{attribute 'linkalways'} 
{attribute 'no_explicit_call' := 'This FB is a CLASS and must be accessed using methods or properties'}
FUNCTION_BLOCK Nci EXTENDS CyclicInstance IMPLEMENTS I_Nci
VAR
	_nciPlc : NciPlc;
END_VAR

PROPERTY _InternalNciPlcRef : REFERENCE TO NciPlc
GET
_InternalNciPlcRef REF= _nciPlc;
END_GET
END_PROPERTY

METHOD AddAxisToGroup
VAR_INPUT
	axis : I_Axis;
	index : UDINT;
	timeout : TIME;
	feedback : REFERENCE TO I_CommandFeedback;
END_VAR
VAR_INST
	pCmd : POINTER TO AddAxisToGroupCommand;
END_VAR
VAR
	_axis : I_Axis;
	_index : UDINT;
	_timeout : TIME;
END_VAR
_axis := axis;
_index := index;
_timeout := timeout;

pCmd := __NEW(AddAxisToGroupCommand(
	nci := THIS^,
	axis := _axis,
	index := _index,
	timeout := _timeout
));

(*
This doesn't work hence the horrible hack with intermediate values

pCmd := __NEW(AddAxisToGroupCommand(
	nci := THIS^,
	axis := axis,
	index := index,
	timeout := timeout
));
*)

pCmd^.Execute(feedback).ThenRelease();
END_METHOD

PROPERTY BlockNumber : UDINT
GET
BlockNumber := ItpGetBlockNumber(THIS^._nciPlc.nciToPlc);
END_GET
END_PROPERTY

METHOD BuildXYGroup
VAR_INPUT
	xAxis : I_Axis;
	yAxis : I_Axis;
	timeout : TIME;
	feedback : REFERENCE TO I_CommandFeedback;
END_VAR
VAR
	null : I_Axis;
END_VAR
BuildXYZGroup(xAxis, yAxis, null, timeout, feedback);
END_METHOD

METHOD BuildXYZGroup
VAR_INPUT
	xAxis : I_Axis;
	yAxis : I_Axis;
	zAxis : I_Axis;
	timeout : TIME;
	feedback : REFERENCE TO I_CommandFeedback;
END_VAR
VAR_INST
	pCmd : POINTER TO BuildXYZGroupCommand;
END_VAR
VAR
	_xAxis : I_Axis;
	_yAxis : I_Axis;
	_zAxis : I_Axis;
	_timeout : TIME;
END_VAR
_xAxis := xAxis;
_yAxis := yAxis;
_zAxis := zAxis;
_timeout := timeout;

pCmd := __NEW(BuildXYZGroupCommand(
	nci := THIS^,
	xAxis := _xAxis,
	yAxis := _yAxis,
	zAxis := _zAxis,
	timeout := _timeout
));

(*
This doesn't work hence the horrible hack with intermediate values

pCmd := __NEW(BuildXYZGroupCommand(
	nci := THIS^,
	xAxis := xAxis,
	yAxis := yAxis,
	zAxis := zAxis,
	timeout := commandTimeout
));
*)

pCmd^.Execute(feedback).ThenRelease();
END_METHOD

PROPERTY ChannelId : UINT
GET
ChannelId := ItpGetChannelId(THIS^._nciPlc.nciToPlc);
END_GET
END_PROPERTY

PROPERTY ChannelType : ChannelType
GET
VAR
	inter : INT;
	pInter : POINTER TO ChannelType;
END_VAR
// Don't know how to do the type conversion with NCIChannelType being strict
inter := ItpGetChannelType(THIS^._nciPlc.nciToPlc);
pInter := ADR(inter);
ChannelType := pInter^;
END_GET
END_PROPERTY

METHOD  CyclicCall
END_METHOD

PROPERTY ErrorId : UDINT
GET
ErrorId := ItpGetError(THIS^._nciPlc.nciToPlc);
END_GET
END_PROPERTY

METHOD GetGroupAxisIds : DWORD
VAR_IN_OUT
	axisIds : ARRAY[1..8] OF DWORD;
END_VAR
GetGroupAxisIds := ItpGetGroupAxisIds(axisIds, THIS^._nciPlc.nciToPlc);
END_METHOD

METHOD GetOverride : LREAL
GetOverride := ItpGetOverridePercent(THIS^._nciPlc.plcToNci);
END_METHOD

PROPERTY GroupId : UDINT
GET
GroupId := ItpGetGroupId(THIS^._nciPlc.nciToPlc);
END_GET
END_PROPERTY

PROPERTY HandshakeableMFunction : INT
GET
HandshakeableMFunction := ItpGetHskMFunc(THIS^._nciPlc.nciToPlc);
END_GET
END_PROPERTY

PROPERTY HasError : BOOL
GET
HasError := ItpHasError(THIS^._nciPlc.nciToPlc);
END_GET
END_PROPERTY

PROPERTY HParam : DINT
GET
HParam := ItpGetHParam(THIS^._nciPlc.nciToPlc);
END_GET
END_PROPERTY

PROPERTY InterpreterState : UDINT
GET
InterpreterState := ItpGetStateInterpreter(THIS^._nciPlc.nciToPlc);
END_GET
END_PROPERTY

PROPERTY IsEstop : BOOL
GET
IsEstop := ItpIsEStopEx(THIS^._nciPlc.nciToPlc);
END_GET
END_PROPERTY

METHOD IsFastMFunctionPresent : BOOL
VAR_INPUT
	functionNumber : INT;
END_VAR
IsFastMFunctionPresent := ItpIsFastMFunc(functionNumber, THIS^._nciPlc.nciToPlc);
END_METHOD

METHOD IsHandshakeableMFunctionPresent : BOOL
IsHandshakeableMFunctionPresent := ItpIsHskMFunc(THIS^._nciPlc.nciToPlc);
END_METHOD

METHOD ReadCyclicLRealParameter : LREAL
VAR_INPUT
	parameterNumber : UINT(1..4);
END_VAR
CASE parameterNumber OF
	1: ReadCyclicLRealParameter := ItpReadCyclicLRealParam1(THIS^._nciPlc.nciToPlc);
	2: ReadCyclicLRealParameter := ItpReadCyclicLRealParam2(THIS^._nciPlc.nciToPlc);
	3: ReadCyclicLRealParameter := ItpReadCyclicLRealParam3(THIS^._nciPlc.nciToPlc);
	4: ReadCyclicLRealParameter := ItpReadCyclicLRealParam4(THIS^._nciPlc.nciToPlc);
END_CASE
END_METHOD

METHOD ReadCyclicUdintParameter : UDINT
VAR_INPUT
	parameterNumber : UINT(1..4);
END_VAR
CASE parameterNumber OF
	1: ReadCyclicUdintParameter := ItpReadCyclicUdintParam1(THIS^._nciPlc.nciToPlc);
	2: ReadCyclicUdintParameter := ItpReadCyclicUdintParam2(THIS^._nciPlc.nciToPlc);
	3: ReadCyclicUdintParameter := ItpReadCyclicUdintParam3(THIS^._nciPlc.nciToPlc);
	4: ReadCyclicUdintParameter := ItpReadCyclicUdintParam4(THIS^._nciPlc.nciToPlc);
END_CASE
END_METHOD

METHOD ReleaseAxis
VAR_INPUT
	axis : I_Axis;
	timeout : TIME;
	feedback : REFERENCE TO I_CommandFeedback;
END_VAR
VAR_INST
	pCmd : POINTER TO ReleaseAxisCommand;
END_VAR
VAR
	_axis : I_Axis;
	_timeout : TIME;
END_VAR
_axis := axis;
_timeout := timeout;

pCmd := __NEW(ReleaseAxisCommand(
	axis := _axis,
	timeout := _timeout
));

(*
This doesn't work hence the horrible hack with intermediate values

pCmd := __NEW(ReleaseAxisCommand(
	axis := axis,
	timeout := timeout
));
*)
pCmd^.Execute(feedback).ThenRelease();
END_METHOD

METHOD ResetGroup
VAR_INPUT
	timeout : TIME;
	feedback : REFERENCE TO I_CommandFeedback;
END_VAR
VAR_INST
	pCmd : POINTER TO ResetGroupCommand;
END_VAR
VAR
	_timeout : TIME;
END_VAR
_timeout := timeout;

pCmd := __NEW(ResetGroupCommand(
	nci := THIS^,
	timeout := _timeout
));

(*
This doesn't work hence the horrible hack with intermediate values

pCmd := __NEW(ResetGroupCommand(
	nci := THIS^,
	timeout := timeout
));
*)

pCmd^.Execute(feedback).ThenRelease();
END_METHOD

METHOD SetOverride : BOOL
VAR_INPUT
	value : LREAL;
END_VAR
SetOverride := ItpSetOverridePercent(value, THIS^._nciPlc.plcToNci);
END_METHOD

PROPERTY SetPathVelocity : LREAL
GET
SetPathVelocity := ItpGetSetPathVelocity(THIS^._nciPlc.nciToPlc);
END_GET
END_PROPERTY

PROPERTY SParam : UINT
GET
SParam := ItpGetSParam(THIS^._nciPlc.nciToPlc);
END_GET
END_PROPERTY

PROPERTY TParam : UINT
GET
TParam := ItpGetTParam(THIS^._nciPlc.nciToPlc);
END_GET
END_PROPERTY

END_FUNCTION_BLOCK

(* stored: Version 1.1.0.1, ProductVersion 3.1.4024.12
   POU Nci: Id {f8cebd7c-fc9e-4bf6-b3ff-461adbfedacc}, SpecialFunc None
   Folder Configuration: Id {64e2e5db-49fe-436d-9103-fcc72122f9b7}
   Folder Internal Properties: Id {157f8ea5-8373-4dfe-9910-0a43152f11e5}
   Folder Methods: Id {25adcca2-5d67-4960-a037-73512035c4aa}
   Folder Properties: Id {5da2c792-bd4d-40c2-8670-e6000f20337d}
   Property _InternalNciPlcRef: Id {22d49991-15d3-421c-a941-a47a723b9637}
   Get Get: Id {779565a3-f0cd-45dc-94f9-cd3182069f1d}
   Method AddAxisToGroup: Id {1ab094d4-4928-4a3d-bd75-9ccaa64be078}
   Property BlockNumber: Id {92b7dfaf-6c64-4bec-af95-15d16a701905}
   Get Get: Id {834fa829-7701-4239-b48a-ed882f001515}
   Method BuildXYGroup: Id {2084a74a-9894-4095-a05c-b558a62448bd}
   Method BuildXYZGroup: Id {7ce7ecfb-d8a2-44cd-86f8-2103482bada6}
   Property ChannelId: Id {34a0a44b-2b1b-4119-a41a-9885bdb3a5b3}
   Get Get: Id {2c6b50fa-e063-45bf-a35f-5d77165c7b4c}
   Property ChannelType: Id {f1398c1a-cd7b-48a7-a865-565888ee9f42}
   Get Get: Id {4ec794f3-f5d0-47c4-aa96-b2c320f82363}
   Method CyclicCall: Id {4ede40d1-7050-4f2d-bfeb-a81bf4477046}
   Property ErrorId: Id {90a95cf4-1833-40d0-b848-d1e1629d9477}
   Get Get: Id {efc9fcf3-a6c2-4566-9265-8dcbe7a5e066}
   Method GetGroupAxisIds: Id {aa1d7dc3-9a02-4f97-9cb7-85dbfd4aa6b9}
   Method GetOverride: Id {a0929981-6171-43dd-957d-687fe4dc1a5d}
   Property GroupId: Id {93889c91-2c81-4f58-8ef3-e41fbc76ada6}
   Get Get: Id {cc900832-7371-46eb-af34-daefcdfde3f2}
   Property HandshakeableMFunction: Id {a2fc5474-1a7f-403a-b555-ae5a827e7fbd}
   Get Get: Id {e43b6f61-6f70-454d-88ea-25be705d3f23}
   Property HasError: Id {aadaec39-bf03-4107-a261-91154fac9f05}
   Get Get: Id {1bc99659-cc6c-4782-9a53-06f9bb48a795}
   Property HParam: Id {a85344b2-d8cc-441b-9fcb-0c3e51d58f2d}
   Get Get: Id {9d73e091-2810-4e52-b9d9-9a704a64cd9a}
   Property InterpreterState: Id {d54ce60d-29f4-4ea2-92ca-5eb3838c56b5}
   Get Get: Id {92dc3f6c-4ce0-4483-a555-8cb59181905b}
   Property IsEstop: Id {184949ff-2e4b-459c-b498-ccae1cd0ceb6}
   Get Get: Id {8635629e-2183-4a4f-95cd-335bdd2b21c3}
   Method IsFastMFunctionPresent: Id {544f6876-a9b1-4ab7-9018-fed31e31baab}
   Method IsHandshakeableMFunctionPresent: Id {cb5e966b-463a-49f2-83fa-9e9198308307}
   Method ReadCyclicLRealParameter: Id {c627ac3e-baa3-4b6d-9895-618922fc341d}
   Method ReadCyclicUdintParameter: Id {e53e0960-4a6b-4031-a73c-d6a592bf35ba}
   Method ReleaseAxis: Id {3f1e7a0d-8dd3-46c7-b807-bbf87effe4df}
   Method ResetGroup: Id {982954cc-7809-4e10-9847-26a8b559aff9}
   Method SetOverride: Id {a0866dab-b495-41bf-b5ac-136f30b3de64}
   Property SetPathVelocity: Id {5ce7e9e2-0f7d-4aca-b58b-c1ee3d559772}
   Get Get: Id {b0cc698d-25e7-4407-9d0f-8707d8bbacd4}
   Property SParam: Id {bc3a4f49-fc7a-46b8-969a-abbbb9aceb9b}
   Get Get: Id {bb9824c6-09f5-4622-be7b-e2a380719954}
   Property TParam: Id {7f42a95f-0912-40d8-a9c5-0689ed9fd19a}
   Get Get: Id {98dab522-f2d4-4aa1-9c14-2c42ec76753e} *)
